FUNCTION_BLOCK Test_LicenceCheck_GetsInValidLicence EXTENDS TUnitTestBase
VAR
END_VAR

METHOD  Execute
VAR_INST
    LicenceCheck : TLicenceCheck(
        LicenceIdAsString      := '{13ae39d9-bbb2-423e-8ace-d2c791a6b0ec}', // 1st digit should be 0
        LicenceName            := 'tcl_BaseLib',
        StopTwinCAT_IfNotValid := FALSE);
END_VAR
IF NOT TestStarted THEN
    LicenceCheck.FB_init(
        bInitRetains            := FALSE,
        bInCopyCode             := FALSE,
        LicenceIdAsString      := '{13ae39d9-bbb2-423e-8ace-d2c791a6b0ec}', // 1st digit should be 0
        LicenceName            := 'tcl_BaseLib',
        StopTwinCAT_IfNotValid := FALSE);
    Test_Started();
END_IF
LicenceCheck();

IF LicenceCheck.CheckComplete THEN
    Assertion.AssertEquals_BOOL(
        Expected := FALSE,
        Actual   := LicenceCheck.IsValid,
        ObjectName := _TestName,
        VariableName  := 'LicenceCheck.IsValid');
    Test_Finished();
END_IF
END_METHOD

END_FUNCTION_BLOCK

(* stored: Version 1.1.0.1, ProductVersion 3.1.4024.3
   POU Test_LicenceCheck_GetsInValidLicence: Id {5a20298c-f10a-0da1-1d93-2960684224ef}, SpecialFunc None
   Method Execute: Id {084dbae0-9c3b-0668-1674-dcdab7bb760f} *)
